Staubli VAL3: start.pgx

program start()
begin
  nPush = 0
  nPop = 0
  nElems = 0
end
